// Mitsubishi GX Works2 project: 공장제어1   PLC: Q03UDV

PROGRAM MAIN
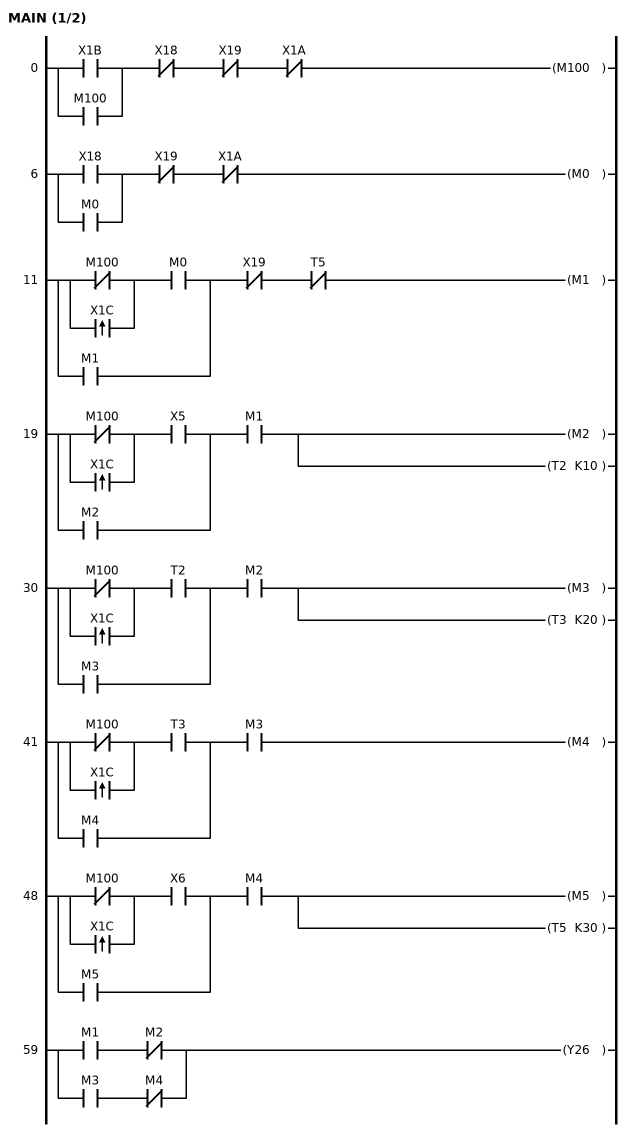
0     LD      X1B
      OR      M100
      ANI     X18
      ANI     X19
      ANI     X1A
      OUT     M100
6     LD      X18
      OR      M0
      ANI     X19
      ANI     X1A
      OUT     M0
11    LDI     M100
      ORP     X1C
      AND     M0
      OR      M1
      ANI     X19
      ANI     T5
      OUT     M1
19    LDI     M100
      ORP     X1C
      AND     X5
      OR      M2
      AND     M1
      OUT     M2
      OUT     T2 K10
30    LDI     M100
      ORP     X1C
      AND     T2
      OR      M3
      AND     M2
      OUT     M3
      OUT     T3 K20
41    LDI     M100
      ORP     X1C
      AND     T3
      OR      M4
      AND     M3
      OUT     M4
48    LDI     M100
      ORP     X1C
      AND     X6
      OR      M5
      AND     M4
      OUT     M5
      OUT     T5 K30
59    LD      M1
      ANI     M2
      LD      M3
      ANI     M4
      ORB
      OUT     Y26
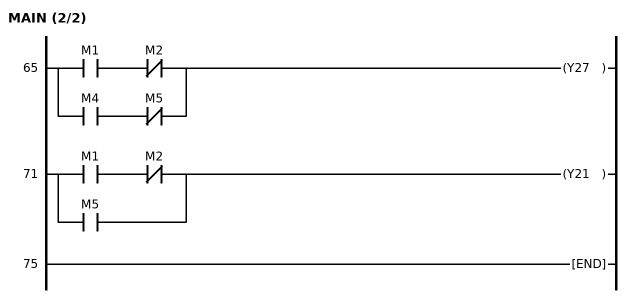
65    LD      M1
      ANI     M2
      LD      M4
      ANI     M5
      ORB
      OUT     Y27
71    LD      M1
      ANI     M2
      OR      M5
      OUT     Y21
75    END
END_PROGRAM
